Fanuc KAREL source: kb00099.KL

-- PROVISIONAL review KL for V940-1; original PC SHA256 cfa0eb04f97cae03810ba273a7bd4c83310b7a558703bcf1491da9f1a7ccb4eb
-- Incomplete behavior may be omitted. Consult companion uncertainty JSON. Do not deploy.
PROGRAM KB00099
%NOLOCKGROUP
VAR
  P1 : STRING[80]
  P2 : STRING[80]
  RESULT : INTEGER
BEGIN
  -- V9_ZERO_TABLE_METADATA_HINT layout=0001; no indexed target words; source/name/runtime held
  -- UNRESOLVED_PC offsets 5-14; opcodes 3F,75
  -- UNRESOLVED_PC offsets 19-28; opcodes 3F,75
  -- UNRESOLVED_PC offsets 33-58; opcodes 27,22,2A,22,2A,76,23
  -- UNRESOLVED_PC offsets 63-67; opcodes 7F
END KB00099
